// Mitsubishi GX Works2 project: 拨片式分拣   PLC: FX2N/FX2NC

PROGRAM MAIN
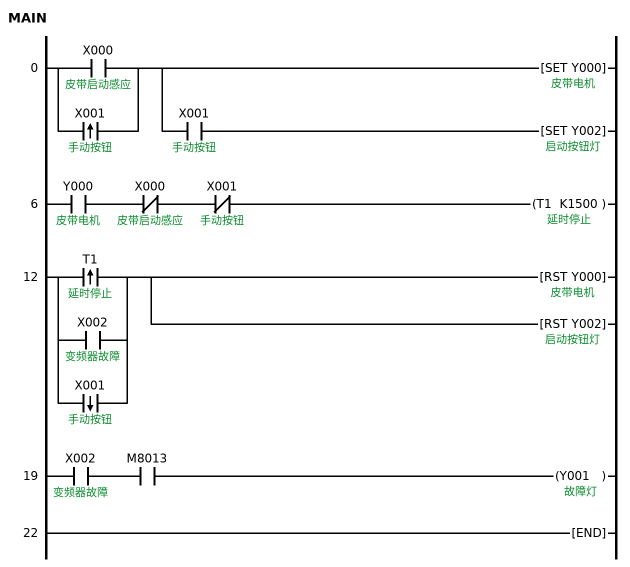
0     LD      X000  ; 皮带启动感应
      ORP     X001  ; 手动按钮
      SET     Y000  ; 皮带电机
      AND     X001  ; 手动按钮
      SET     Y002  ; 启动按钮灯
6     LD      Y000  ; 皮带电机
      ANI     X000  ; 皮带启动感应
      ANI     X001  ; 手动按钮
      OUT     T1 K1500  ; 延时停止
12    LDP     T1  ; 延时停止
      OR      X002  ; 变频器故障
      ORF     X001  ; 手动按钮
      RST     Y000  ; 皮带电机
      RST     Y002  ; 启动按钮灯
19    LD      X002  ; 变频器故障
      AND     M8013
      OUT     Y001  ; 故障灯
22    END
END_PROGRAM
